// TIA Portal V17 export
// export: Created 2025-03-13T10:29:39.2691686Z, ExportSetting WithDefaults, DisplayName Totally Integrated Automation Portal, DisplayVersion V17 Update 8, DisplayName TIA Portal Openness, DisplayVersion V17 Update 8, DisplayName TIA Portal Version Control Interface, DisplayVersion V17, DisplayName SINAMICS Startdrive Advanced, DisplayVersion V17 SP2, DisplayName SINAMICS Startdrive G110M, G120, G120C, G120D, G120P, G115D, DisplayVersion V17 SP2, DisplayName SINAMICS Startdrive G130, G150, S120, S150, SINAMICS MV, S210, DisplayVersion V17 SP2, DisplayName STEP 7 Professional, DisplayVersion V17 Update 8, DisplayName SINUMERIK ONE STEP 7 Toolbox, DisplayVersion V17 Update 12, DisplayName SINUMERIK 840D sl STEP 7 Toolbox, DisplayVersion V17 Update 12, DisplayName STEP 7 Safety, DisplayVersion V17 Update 6, DisplayName WinCC Advanced, DisplayVersion V17 Update 8
FUNCTION_BLOCK "Main_Safety_RTG1"   // FB1010, F_LAD
{ S7_Optimized_Access := 'TRUE' }
VERSION : 0.1
// stored: AutoNumber false, IsIECCheckEnabled false, UDAEnableTagReadback false
   VAR
      ACK_GL_Instance : ACK_GL;
   END_VAR
BEGIN

REGION Network 1: RECEIVE SAFE I/O FROM NCU
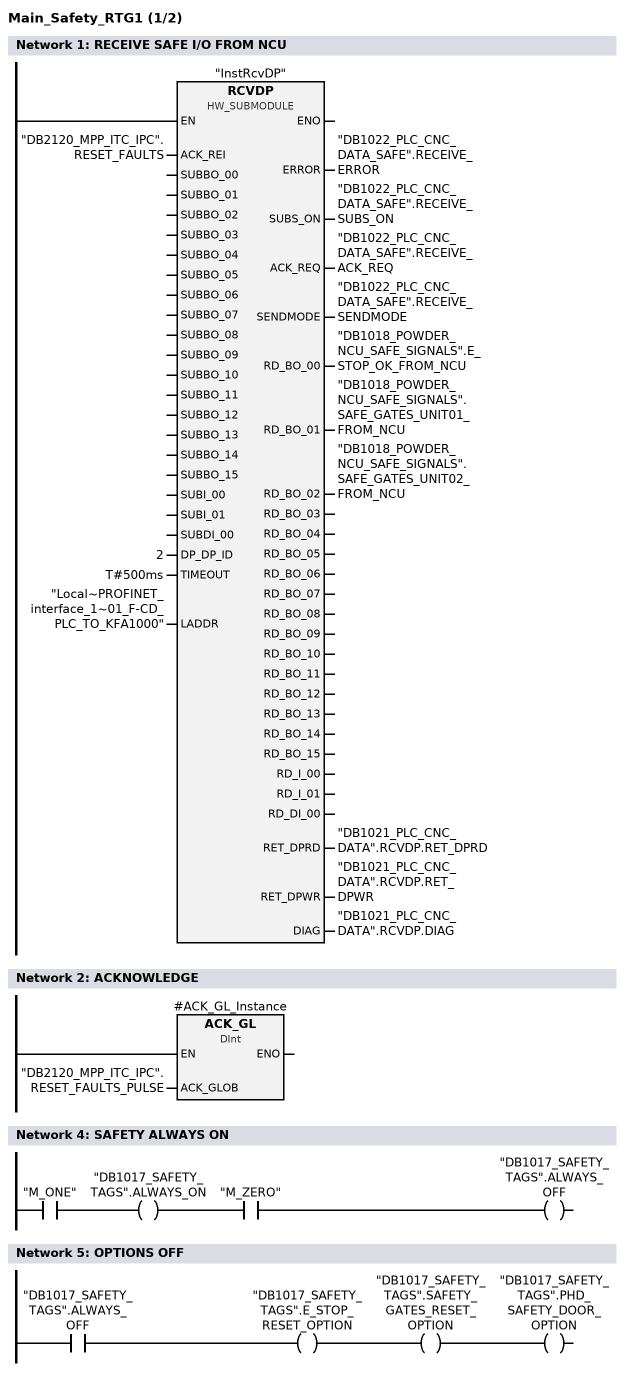
   RUNG wire#powerrail
      { S7_Templates := "laddr_type := HW_SUBMODULE" } "InstRcvDP".RCVDP(ACK_REI := "DB2120_MPP_ITC_IPC".RESET_FAULTS, SUBBO_00 :=, SUBBO_01 :=, SUBBO_02 :=, SUBBO_03 :=, SUBBO_04 :=, SUBBO_05 :=, SUBBO_06 :=, SUBBO_07 :=, SUBBO_08 :=, SUBBO_09 :=, SUBBO_10 :=, SUBBO_11 :=, SUBBO_12 :=, SUBBO_13 :=, SUBBO_14 :=, SUBBO_15 :=, SUBI_00 :=, SUBI_01 :=, SUBDI_00 :=, DP_DP_ID := 2, TIMEOUT := T#500ms, LADDR := "Local~PROFINET_interface_1~01_F-CD_PLC_TO_KFA1000", ERROR => "DB1022_PLC_CNC_DATA_SAFE".RECEIVE_ERROR, SUBS_ON => "DB1022_PLC_CNC_DATA_SAFE".RECEIVE_SUBS_ON, ACK_REQ => "DB1022_PLC_CNC_DATA_SAFE".RECEIVE_ACK_REQ, SENDMODE => "DB1022_PLC_CNC_DATA_SAFE".RECEIVE_SENDMODE, RD_BO_00 => "DB1018_POWDER_NCU_SAFE_SIGNALS".E_STOP_OK_FROM_NCU, RD_BO_01 => "DB1018_POWDER_NCU_SAFE_SIGNALS".SAFE_GATES_UNIT01_FROM_NCU, RD_BO_02 => "DB1018_POWDER_NCU_SAFE_SIGNALS".SAFE_GATES_UNIT02_FROM_NCU, RD_BO_03 =>, RD_BO_04 =>, RD_BO_05 =>, RD_BO_06 =>, RD_BO_07 =>, RD_BO_08 =>, RD_BO_09 =>, RD_BO_10 =>, RD_BO_11 =>, RD_BO_12 =>, RD_BO_13 =>, RD_BO_14 =>, RD_BO_15 =>, RD_I_00 =>, RD_I_01 =>, RD_DI_00 =>, RET_DPRD => "DB1021_PLC_CNC_DATA".RCVDP.RET_DPRD, RET_DPWR => "DB1021_PLC_CNC_DATA".RCVDP.RET_DPWR, DIAG => "DB1021_PLC_CNC_DATA".RCVDP.DIAG)
   END_RUNG
   // the same network as SCL:
   "InstRcvDP"(ACK_REI := "DB2120_MPP_ITC_IPC".RESET_FAULTS,   // RCVDP
               DP_DP_ID := 2,
               TIMEOUT := T#500ms,
               LADDR := "Local~PROFINET_interface_1~01_F-CD_PLC_TO_KFA1000",
               ERROR => "DB1022_PLC_CNC_DATA_SAFE".RECEIVE_ERROR,
               SUBS_ON => "DB1022_PLC_CNC_DATA_SAFE".RECEIVE_SUBS_ON,
               ACK_REQ => "DB1022_PLC_CNC_DATA_SAFE".RECEIVE_ACK_REQ,
               SENDMODE => "DB1022_PLC_CNC_DATA_SAFE".RECEIVE_SENDMODE,
               RD_BO_00 => "DB1018_POWDER_NCU_SAFE_SIGNALS".E_STOP_OK_FROM_NCU,
               RD_BO_01 => "DB1018_POWDER_NCU_SAFE_SIGNALS".SAFE_GATES_UNIT01_FROM_NCU,
               RD_BO_02 => "DB1018_POWDER_NCU_SAFE_SIGNALS".SAFE_GATES_UNIT02_FROM_NCU,
               RET_DPRD => "DB1021_PLC_CNC_DATA".RCVDP.RET_DPRD,
               RET_DPWR => "DB1021_PLC_CNC_DATA".RCVDP.RET_DPWR,
               DIAG => "DB1021_PLC_CNC_DATA".RCVDP.DIAG);
END_REGION

REGION Network 2: ACKNOWLEDGE
   RUNG wire#powerrail
      { S7_Templates := "codedbool_type := DInt" } #ACK_GL_Instance.ACK_GL(ACK_GLOB := "DB2120_MPP_ITC_IPC".RESET_FAULTS_PULSE)
   END_RUNG
   // the same network as SCL:
   #ACK_GL_Instance(ACK_GLOB := "DB2120_MPP_ITC_IPC".RESET_FAULTS_PULSE);   // ACK_GL
END_REGION

REGION Network 4: SAFETY ALWAYS ON
   RUNG wire#powerrail
      Contact( "M_ONE" )
      Coil( "DB1017_SAFETY_TAGS".ALWAYS_ON )
      Contact( "M_ZERO" )
      Coil( "DB1017_SAFETY_TAGS".ALWAYS_OFF )
   END_RUNG
   // the same network as SCL:
   "DB1017_SAFETY_TAGS".ALWAYS_ON := "M_ONE";
   "DB1017_SAFETY_TAGS".ALWAYS_OFF := "M_ONE" AND "M_ZERO";
END_REGION

REGION Network 5: OPTIONS OFF
   RUNG wire#powerrail
      Contact( "DB1017_SAFETY_TAGS".ALWAYS_OFF )
      Coil( "DB1017_SAFETY_TAGS".E_STOP_RESET_OPTION )
      Coil( "DB1017_SAFETY_TAGS".SAFETY_GATES_RESET_OPTION )
      Coil( "DB1017_SAFETY_TAGS".PHD_SAFETY_DOOR_OPTION )
   END_RUNG
   // the same network as SCL:
   "DB1017_SAFETY_TAGS".E_STOP_RESET_OPTION := "DB1017_SAFETY_TAGS".ALWAYS_OFF;
   "DB1017_SAFETY_TAGS".SAFETY_GATES_RESET_OPTION := "DB1017_SAFETY_TAGS".ALWAYS_OFF;
   "DB1017_SAFETY_TAGS".PHD_SAFETY_DOOR_OPTION := "DB1017_SAFETY_TAGS".ALWAYS_OFF;
END_REGION

REGION Network 6: OPTIONS ON
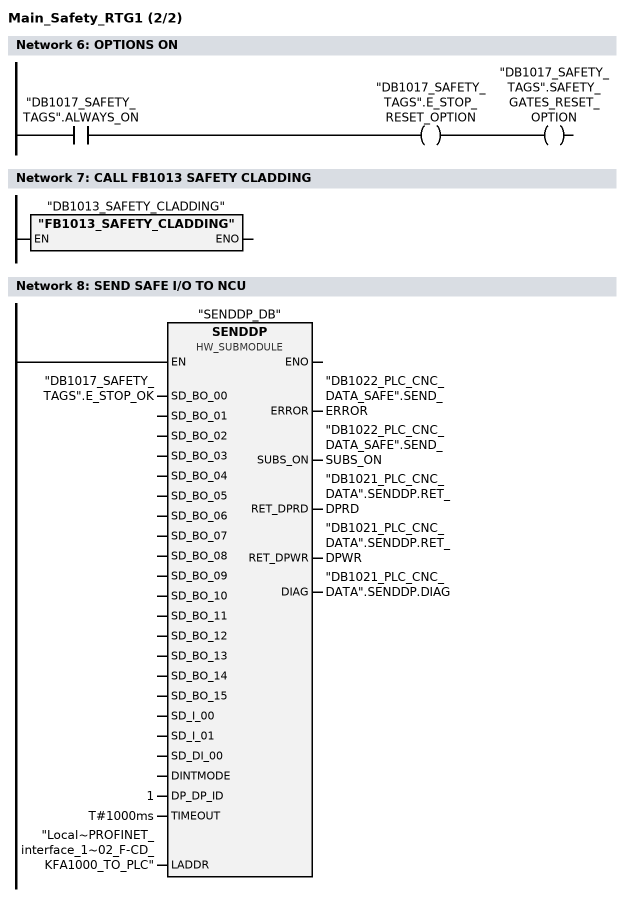
   RUNG wire#powerrail
      Contact( "DB1017_SAFETY_TAGS".ALWAYS_ON )
      Coil( "DB1017_SAFETY_TAGS".E_STOP_RESET_OPTION )
      Coil( "DB1017_SAFETY_TAGS".SAFETY_GATES_RESET_OPTION )
   END_RUNG
   // the same network as SCL:
   "DB1017_SAFETY_TAGS".E_STOP_RESET_OPTION := "DB1017_SAFETY_TAGS".ALWAYS_ON;
   "DB1017_SAFETY_TAGS".SAFETY_GATES_RESET_OPTION := "DB1017_SAFETY_TAGS".ALWAYS_ON;
END_REGION

REGION Network 7: CALL FB1013 SAFETY CLADDING
   RUNG wire#powerrail
      "DB1013_SAFETY_CLADDING"()
   END_RUNG
   // the same network as SCL:
   "DB1013_SAFETY_CLADDING"();   // "FB1013_SAFETY_CLADDING"
END_REGION

REGION Network 8: SEND SAFE I/O TO NCU
   RUNG wire#powerrail
      { S7_Templates := "laddr_type := HW_SUBMODULE" } "SENDDP_DB".SENDDP(SD_BO_00 := "DB1017_SAFETY_TAGS".E_STOP_OK, SD_BO_01 :=, SD_BO_02 :=, SD_BO_03 :=, SD_BO_04 :=, SD_BO_05 :=, SD_BO_06 :=, SD_BO_07 :=, SD_BO_08 :=, SD_BO_09 :=, SD_BO_10 :=, SD_BO_11 :=, SD_BO_12 :=, SD_BO_13 :=, SD_BO_14 :=, SD_BO_15 :=, SD_I_00 :=, SD_I_01 :=, SD_DI_00 :=, DINTMODE :=, DP_DP_ID := 1, TIMEOUT := T#1000ms, LADDR := "Local~PROFINET_interface_1~02_F-CD_KFA1000_TO_PLC", ERROR => "DB1022_PLC_CNC_DATA_SAFE".SEND_ERROR, SUBS_ON => "DB1022_PLC_CNC_DATA_SAFE".SEND_SUBS_ON, RET_DPRD => "DB1021_PLC_CNC_DATA".SENDDP.RET_DPRD, RET_DPWR => "DB1021_PLC_CNC_DATA".SENDDP.RET_DPWR, DIAG => "DB1021_PLC_CNC_DATA".SENDDP.DIAG)
   END_RUNG
   // the same network as SCL:
   "SENDDP_DB"(SD_BO_00 := "DB1017_SAFETY_TAGS".E_STOP_OK,   // SENDDP
               DP_DP_ID := 1,
               TIMEOUT := T#1000ms,
               LADDR := "Local~PROFINET_interface_1~02_F-CD_KFA1000_TO_PLC",
               ERROR => "DB1022_PLC_CNC_DATA_SAFE".SEND_ERROR,
               SUBS_ON => "DB1022_PLC_CNC_DATA_SAFE".SEND_SUBS_ON,
               RET_DPRD => "DB1021_PLC_CNC_DATA".SENDDP.RET_DPRD,
               RET_DPWR => "DB1021_PLC_CNC_DATA".SENDDP.RET_DPWR,
               DIAG => "DB1021_PLC_CNC_DATA".SENDDP.DIAG);
END_REGION
END_FUNCTION_BLOCK
